(* PLC project CHL-DZ-BJDX-11 宁波数字孪生（东方理工）研究院制备薄层色谱全自动化工作站_Old_InoProShop(V1.9.1.6).project, Inovance company InoProShop(V1.9.1.6) InoProShop(V1.9.1.6) *)
(* stored: creationDateTime 2026-06-16T17:56:22.3681085, modificationDateTime 2026-06-04T10:59:46 *)

PROGRAM PLC_Cyinder_气缸动作
  VAR
    cylinder_0 : FB_cylinder;
    cylinder_1 : FB_cylinder;
    cylinder_2 : FB_cylinder;
    cylinder_3 : FB_cylinder;
    cylinder_4 : FB_cylinder;
    cylinder_5 : FB_cylinder;
    cylinder_6 : FB_cylinder;
    cylinder_7 : FB_cylinder;
    cylinder_8 : FB_cylinder;
    cylinder_9 : FB_cylinder;
    cylinder_10 : FB_cylinder;
    cylinder_11 : FB_cylinder;
    cylinder_12 : FB_cylinder;
    cylinder_13 : FB_cylinder;
    cylinder_14 : FB_cylinder;
    cylinder_15 : FB_cylinder;
    cylinder_16 : FB_cylinder;
    cylinder_17 : FB_cylinder;
    cylinder_18 : FB_cylinder;
    cylinder_19 : FB_cylinder;
    cylinder_20 : FB_cylinder;
    cylinder_21 : FB_cylinder;
    cylinder_22 : FB_cylinder;
    cylinder_23 : FB_cylinder;
    cylinder_24 : FB_cylinder;
    cylinder_25 : FB_cylinder;
    cylinder_26 : FB_cylinder;
    cylinder_27 : FB_cylinder;
    cylinder_28 : FB_cylinder;
    cylinder_29 : FB_cylinder;
    cylinder_30 : FB_cylinder;
    cylinder_31 : FB_cylinder;
    cylinder_32 : FB_cylinder;
    cylinder_33 : FB_cylinder;
    cylinder_34 : FB_cylinder;
    cylinder_35 : FB_cylinder;
    cylinder_36 : FB_cylinder;
    cylinder_37 : FB_cylinder;
    cylinder_38 : FB_cylinder;
    cylinder_39 : FB_cylinder;
    cylinder_40 : FB_cylinder;
    cylinder_41 : FB_cylinder;
    cylinder_42 : FB_cylinder;
    cylinder_43 : FB_cylinder;
    cylinder_44 : FB_cylinder;
    cylinder_45 : FB_cylinder;
    cylinder_46 : FB_cylinder;
    cylinder_47 : FB_cylinder;
    cylinder_48 : FB_cylinder;
    cylinder_49 : FB_cylinder;
    cylinder_50 : FB_cylinder;
  END_VAR

            //气缸动作
//展缸1气缸1
cylinder_0(
    xManualRetract := , 
    xAutoRetract := , 
    yValve2 => , 
    cylinder_type := 0, 

	xManualAuto:=ManualAuto  , 
	xManualExtend:=展缸1气缸1手动 , 
	xAutoExtend:= 展缸1气缸1自动, 
	xReset:=复位  , 
	xPosExtend:= 展缸1气缸1原点, 
	xPosRetract:= 展缸1气缸1动点 , 
	tTimeout:= T#5S, 
	yValve1=> 展缸1气缸1 , 
	bAlarm=> cyinderAlarm.0);
//展缸1气缸2
cylinder_1(
    xManualRetract := , 
    xAutoRetract := , 
    yValve2 => , 
    cylinder_type :=0 , 

	xManualAuto:=ManualAuto  , 
	xManualExtend:=展缸1气缸2手动 , 
	xAutoExtend:= 展缸1气缸2自动, 
	xReset:=复位  , 
	xPosExtend:= 展缸1气缸2原点, 
	xPosRetract:= 展缸1气缸2动点 , 
	tTimeout:= T#5S, 
	yValve1=> 展缸1气缸2, 
	bAlarm=> cyinderAlarm.1);
//展缸1气缸3
cylinder_2(
    xManualRetract := , 
    xAutoRetract := , 
    yValve2 => , 
    cylinder_type := 0, 

	xManualAuto:=ManualAuto  , 
	xManualExtend:=展缸1气缸3手动 , 
	xAutoExtend:= 展缸1气缸3自动, 
	xReset:=复位  , 
	xPosExtend:= 展缸1气缸3原点, 
	xPosRetract:= 展缸1气缸3动点 , 
	tTimeout:= T#5S, 
	yValve1=> 展缸1气缸3, 
	bAlarm=> cyinderAlarm.2);
//展缸1气缸4
cylinder_3(
    xManualRetract := , 
    xAutoRetract := , 
    yValve2 => , 
    cylinder_type :=0 , 

	xManualAuto:=ManualAuto  , 
	xManualExtend:=展缸1气缸4手动 , 
	xAutoExtend:= 展缸1气缸4自动, 
	xReset:=复位  , 
	xPosExtend:= 展缸1气缸4原点, 
	xPosRetract:= 展缸1气缸4动点 , 
	tTimeout:= T#5S, 
	yValve1=> 展缸1气缸4, 
	bAlarm=> cyinderAlarm.3);
//展缸2气缸1
cylinder_4(
    xManualRetract := , 
    xAutoRetract := , 
    yValve2 => , 
    cylinder_type := 0, 

	xManualAuto:=ManualAuto  , 
	xManualExtend:=展缸2气缸1手动 , 
	xAutoExtend:= 展缸2气缸1自动, 
	xReset:=复位  , 
	xPosExtend:= 展缸2气缸1原点, 
	xPosRetract:= 展缸2气缸1动点 , 
	tTimeout:= T#5S, 
	yValve1=> 展缸2气缸1, 
	bAlarm=> cyinderAlarm.4);
//展缸2气缸2
cylinder_5(
    xManualRetract := , 
    xAutoRetract := , 
    yValve2 => , 
    cylinder_type :=0 , 

	xManualAuto:=ManualAuto  , 
	xManualExtend:=展缸2气缸2手动 , 
	xAutoExtend:= 展缸2气缸2自动, 
	xReset:=复位  , 
	xPosExtend:= 展缸2气缸2原点, 
	xPosRetract:= 展缸2气缸2动点 , 
	tTimeout:= T#5S, 
	yValve1=> 展缸2气缸2, 
	bAlarm=> cyinderAlarm.5);
//展缸2气缸3
cylinder_6(
    xManualRetract := , 
    xAutoRetract := , 
    yValve2 => , 
    cylinder_type := 0, 

	xManualAuto:=ManualAuto  , 
	xManualExtend:=展缸2气缸3手动 , 
	xAutoExtend:= 展缸2气缸3自动, 
	xReset:=复位  , 
	xPosExtend:= 展缸2气缸3原点, 
	xPosRetract:= 展缸2气缸3动点 , 
	tTimeout:= T#5S, 
	yValve1=> 展缸2气缸3, 
	bAlarm=> cyinderAlarm.6);
//展缸2气缸4
cylinder_7(
    xManualRetract := , 
    xAutoRetract := , 
    yValve2 => , 
    cylinder_type := 0, 

	xManualAuto:=ManualAuto  , 
	xManualExtend:=展缸2气缸4手动 , 
	xAutoExtend:= 展缸2气缸4自动, 
	xReset:=复位  , 
	xPosExtend:= 展缸2气缸4原点, 
	xPosRetract:= 展缸2气缸4动点 , 
	tTimeout:= T#5S, 
	yValve1=> 展缸2气缸4, 
	bAlarm=> cyinderAlarm.7);
//大真空泵
cylinder_8(
    xManualRetract := , 
    xAutoRetract := , 
    yValve2 => , 
    cylinder_type :=0 , 

	xManualAuto:=ManualAuto  , 
	xManualExtend:= 大真空泵手动, 
	xAutoExtend:= 大真空泵自动, 
	xReset:=复位  , 
	xPosExtend:= , 
	xPosRetract:=  , 
	tTimeout:= , 
	yValve1=> 大真空泵, 
	bAlarm=> );
//收集平台下压气缸
cylinder_9(
    xManualRetract := , 
    xAutoRetract := , 
    yValve2 => , 
    cylinder_type := 0, 

	xManualAuto:=ManualAuto  , 
	xManualExtend:= 收集下压气缸手动, 
	xAutoExtend:= 收集下压气缸自动, 
	xReset:=复位  , 
	xPosExtend:=收集平台下压气缸原点 , 
	xPosRetract:= 收集下压气缸手动 OR 收集下压气缸自动, 
	tTimeout:= T#5S, 
	yValve1=> 收集下压气缸 , 
	bAlarm=> cyinderAlarm.8);
//收集平台夹持气缸
cylinder_10(
    xManualRetract := , 
    xAutoRetract := , 
    yValve2 => , 
    cylinder_type := 0, 

	xManualAuto:=ManualAuto  , 
	xManualExtend:= 收集夹持气缸手动, 
	xAutoExtend:= 收集夹持气缸自动, 
	xReset:=复位  , 
	xPosExtend:=收集平台夹持气缸原点 , 
	xPosRetract:= 收集平台夹持气缸动点, 
	tTimeout:= T#5S, 
	yValve1=> 收集夹持气缸  , 
	bAlarm=> cyinderAlarm.9);	
//收集平台升降气缸
cylinder_11(
    xManualRetract := , 
    xAutoRetract := , 
    yValve2 => , 
    cylinder_type := 0, 

	xManualAuto:=ManualAuto  , 
	xManualExtend:= 收集升降气缸手动, 
	xAutoExtend:= 收集升降气缸自动, 
	xReset:=复位  , 
	xPosExtend:=收集平台升降气缸原点 , 
	xPosRetract:= 收集平台升降气缸动点, 
	tTimeout:= T#5S, 
	yValve1=> 收集升降气缸   , 
	bAlarm=> cyinderAlarm.10);	
//收集平台伸缩气缸
cylinder_12(
    xManualRetract := , 
    xAutoRetract := , 
    yValve2 => , 
    cylinder_type :=0 , 

	xManualAuto:=ManualAuto  , 
	xManualExtend:= 收集伸缩气缸手动, 
	xAutoExtend:= 收集伸缩气缸自动, 
	xReset:=复位, 
	xPosExtend:=收集平台推出气缸原点, 
	xPosRetract:= 收集平台推出气缸动点, 
	tTimeout:= T#5S, 
	yValve1=> 收集伸缩气缸, 
	bAlarm=> cyinderAlarm.11);		
//刮板拍照遮光气缸
cylinder_13(
    xManualRetract := , 
    xAutoRetract := , 
    yValve2 => , 
    cylinder_type :=0 , 

	xManualAuto:=ManualAuto  , 
	xManualExtend:= 刮板拍照遮光气缸手动, 
	xAutoExtend:=刮板拍照遮光气缸自动 , 
	xReset:=复位  , 
	xPosExtend:=刮板拍照遮光气缸上位 , 
	xPosRetract:= 刮板拍照遮光气缸下位, 
	tTimeout:= T#5S, 
	yValve1=>  刮板拍照遮光气缸, 
	bAlarm=> cyinderAlarm.12);		
//刮板拍照旋转气缸
cylinder_14(
    xManualRetract := , 
    xAutoRetract := , 
    yValve2 => , 
    cylinder_type := 0, 

	xManualAuto:=ManualAuto  , 
	xManualExtend:= 刮板拍照旋转气缸手动 AND 刮板轴9XDATE.fActPos>330, 
	xAutoExtend:=刮板拍照旋转气缸自动 , 
	xReset:=复位  , 
	xPosExtend:=刮板拍照旋转气缸原点  , 
	xPosRetract:= 刮板拍照旋转气缸动点, 
	tTimeout:= T#5S, 
	yValve1=>  刮板拍照旋转气缸   , 
	bAlarm=> cyinderAlarm.13);		
//刮板拍照下压气缸
cylinder_15(
    xManualRetract := , 
    xAutoRetract := , 
    yValve2 => , 
    cylinder_type := 0, 

	xManualAuto:=ManualAuto  , 
	xManualExtend:= 刮板拍照下压气缸手动, 
	xAutoExtend:=刮板拍照下压气缸自动 , 
	xReset:=复位  , 
	xPosExtend:=刮板拍照下压气缸上位, 
	xPosRetract:=刮板拍照下压气缸手动 OR 刮板拍照下压气缸自动 , 
	tTimeout:= T#5S, 
	yValve1=>  刮板拍照下压气缸, 
	bAlarm=> cyinderAlarm.14);
//展缸1进液电池阀1
cylinder_17(
    xManualRetract := , 
    xAutoRetract := , 
    yValve2 => , 
    cylinder_type :=0 , 

	xManualAuto:=ManualAuto  , 
	xManualExtend:= 展缸1进液电池阀1手动, 
	xAutoExtend:= 展缸1进液电池阀1自动, 
	xReset:=复位  , 
	xPosExtend:=   , 
	xPosRetract:= , 
	tTimeout:= , 
	yValve1=> 展缸1进液电池阀1, 
	bAlarm=> );	
//展缸1进液电池阀2
cylinder_18(
    xManualRetract := , 
    xAutoRetract := , 
    yValve2 => , 
    cylinder_type := 0, 

	xManualAuto:=ManualAuto  , 
	xManualExtend:= 展缸1进液电池阀2手动, 
	xAutoExtend:= 展缸1进液电池阀2自动, 
	xReset:=复位  , 
	xPosExtend:=   , 
	xPosRetract:= , 
	tTimeout:= , 
	yValve1=> 展缸1进液电池阀2, 
	bAlarm=> );	
//展缸1进液电池阀3
cylinder_19(
    xManualRetract := , 
    xAutoRetract := , 
    yValve2 => , 
    cylinder_type := 0, 

	xManualAuto:=ManualAuto  , 
	xManualExtend:= 展缸1进液电池阀3手动, 
	xAutoExtend:= 展缸1进液电池阀3自动, 
	xReset:=复位  , 
	xPosExtend:=   , 
	xPosRetract:= , 
	tTimeout:= , 
	yValve1=> 展缸1进液电池阀3, 
	bAlarm=> );	
//展缸1进液电池阀4
cylinder_20(
    xManualRetract := , 
    xAutoRetract := , 
    yValve2 => , 
    cylinder_type := 0, 

	xManualAuto:=ManualAuto  , 
	xManualExtend:= 展缸1进液电池阀4手动, 
	xAutoExtend:= 展缸1进液电池阀4自动, 
	xReset:=复位  , 
	xPosExtend:=   , 
	xPosRetract:= , 
	tTimeout:= , 
	yValve1=> 展缸1进液电池阀4, 
	bAlarm=> );	
//展缸1排液电池阀1
cylinder_21(
    xManualRetract := , 
    xAutoRetract := , 
    yValve2 => , 
    cylinder_type := 0, 

	xManualAuto:=ManualAuto  , 
	xManualExtend:= 展缸1排液电池阀1手动, 
	xAutoExtend:= 展缸1排液电池阀1自动, 
	xReset:=复位  , 
	xPosExtend:=   , 
	xPosRetract:= , 
	tTimeout:= , 
	yValve1=> 展缸1排液电池阀1, 
	bAlarm=> );	
//展缸1排液电池阀2
cylinder_22(
    xManualRetract := , 
    xAutoRetract := , 
    yValve2 => , 
    cylinder_type :=0 , 

	xManualAuto:=ManualAuto  , 
	xManualExtend:= 展缸1排液电池阀2手动, 
	xAutoExtend:= 展缸1排液电池阀2自动, 
	xReset:=复位  , 
	xPosExtend:=   , 
	xPosRetract:= , 
	tTimeout:= , 
	yValve1=> 展缸1排液电池阀2, 
	bAlarm=> );	
//展缸1排液电池阀3
cylinder_23(
    xManualRetract := , 
    xAutoRetract := , 
    yValve2 => , 
    cylinder_type :=0 , 

	xManualAuto:=ManualAuto, 
	xManualExtend:= 展缸1排液电池阀3手动, 
	xAutoExtend:= 展缸1排液电池阀3自动, 
	xReset:=复位  , 
	xPosExtend:=   , 
	xPosRetract:= , 
	tTimeout:= , 
	yValve1=> 展缸1排液电池阀3, 
	bAlarm=> );	
//展缸1排液电池阀4
cylinder_24(
    xManualRetract := , 
    xAutoRetract := , 
    yValve2 => , 
    cylinder_type := 0, 

	xManualAuto:=ManualAuto, 
	xManualExtend:= 展缸1排液电池阀4手动, 
	xAutoExtend:= 展缸1排液电池阀4自动, 
	xReset:=复位  , 
	xPosExtend:=   , 
	xPosRetract:= , 
	tTimeout:= , 
	yValve1=> 展缸1排液电池阀4, 
	bAlarm=> );	
//展缸1吹气电池阀1
cylinder_25(
    xManualRetract := , 
    xAutoRetract := , 
    yValve2 => , 
    cylinder_type := 0, 

	xManualAuto:=ManualAuto, 
	xManualExtend:= 展缸1吹气电池阀1手动, 
	xAutoExtend:= 展缸1吹气电池阀1自动, 
	xReset:=复位  , 
	xPosExtend:=   , 
	xPosRetract:= , 
	tTimeout:= , 
	yValve1=> 展缸1吹气电池阀1, 
	bAlarm=> );	
//展缸1吹气电池阀2
cylinder_26(
    xManualRetract := , 
    xAutoRetract := , 
    yValve2 => , 
    cylinder_type := 0, 

	xManualAuto:=ManualAuto, 
	xManualExtend:= 展缸1吹气电池阀2手动, 
	xAutoExtend:= 展缸1吹气电池阀2自动, 
	xReset:=复位  , 
	xPosExtend:=   , 
	xPosRetract:= , 
	tTimeout:= , 
	yValve1=> 展缸1吹气电池阀2, 
	bAlarm=> );	
//展缸1吹气电池阀3
cylinder_27(
    xManualRetract := , 
    xAutoRetract := , 
    yValve2 => , 
    cylinder_type := 0, 

	xManualAuto:=ManualAuto  , 
	xManualExtend:= 展缸1吹气电池阀3手动, 
	xAutoExtend:= 展缸1吹气电池阀3自动, 
	xReset:=复位  , 
	xPosExtend:=   , 
	xPosRetract:= , 
	tTimeout:= , 
	yValve1=> 展缸1吹气电池阀3, 
	bAlarm=> );	
//展缸1吹气电池阀4
cylinder_28(
    xManualRetract := , 
    xAutoRetract := , 
    yValve2 => , 
    cylinder_type := 0, 

	xManualAuto:=ManualAuto, 
	xManualExtend:= 展缸1吹气电池阀4手动, 
	xAutoExtend:= 展缸1吹气电池阀4自动, 
	xReset:=复位  , 
	xPosExtend:=   , 
	xPosRetract:= , 
	tTimeout:= , 
	yValve1=> 展缸1吹气电池阀4, 
	bAlarm=> );	
//展缸2进液电池阀1
cylinder_29(
    xManualRetract := , 
    xAutoRetract := , 
    yValve2 => , 
    cylinder_type := 0, 

	xManualAuto:=ManualAuto, 
	xManualExtend:= 展缸2进液电池阀1手动, 
	xAutoExtend:= 展缸2进液电池阀1自动, 
	xReset:=复位  , 
	xPosExtend:=   , 
	xPosRetract:= , 
	tTimeout:= , 
	yValve1=> 展缸2进液电池阀1, 
	bAlarm=> );	
//展缸2进液电池阀2
cylinder_30(
    xManualRetract := , 
    xAutoRetract := , 
    yValve2 => , 
    cylinder_type := 0, 

	xManualAuto:=ManualAuto, 
	xManualExtend:= 展缸2进液电池阀2手动, 
	xAutoExtend:= 展缸2进液电池阀2自动, 
	xReset:=复位  , 
	xPosExtend:=   , 
	xPosRetract:= , 
	tTimeout:= , 
	yValve1=> 展缸2进液电池阀2, 
	bAlarm=> );	
//展缸2进液电池阀3
cylinder_31(
    xManualRetract := , 
    xAutoRetract := , 
    yValve2 => , 
    cylinder_type := 0, 

	xManualAuto:=ManualAuto, 
	xManualExtend:= 展缸2进液电池阀3手动, 
	xAutoExtend:= 展缸2进液电池阀3自动, 
	xReset:=复位  , 
	xPosExtend:=   , 
	xPosRetract:= , 
	tTimeout:= , 
	yValve1=> 展缸2进液电池阀3, 
	bAlarm=> );	
//展缸2进液电池阀4
cylinder_32(
    xManualRetract := , 
    xAutoRetract := , 
    yValve2 => , 
    cylinder_type := 0, 

	xManualAuto:=ManualAuto, 
	xManualExtend:= 展缸2进液电池阀4手动, 
	xAutoExtend:= 展缸2进液电池阀4自动, 
	xReset:=复位  , 
	xPosExtend:=   , 
	xPosRetract:= , 
	tTimeout:= , 
	yValve1=> 展缸2进液电池阀4, 
	bAlarm=> );	
//展缸2排液电池阀1
cylinder_33(
    xManualRetract := , 
    xAutoRetract := , 
    yValve2 => , 
    cylinder_type := 0, 

	xManualAuto:=ManualAuto, 
	xManualExtend:= 展缸2排液电池阀1手动, 
	xAutoExtend:= 展缸2排液电池阀1自动, 
	xReset:=复位  , 
	xPosExtend:=   , 
	xPosRetract:= , 
	tTimeout:= , 
	yValve1=> 展缸2排液电池阀1, 
	bAlarm=> );	
//展缸2排液电池阀2
cylinder_34(
    xManualRetract := , 
    xAutoRetract := , 
    yValve2 => , 
    cylinder_type := 0, 

	xManualAuto:=ManualAuto, 
	xManualExtend:= 展缸2排液电池阀2手动, 
	xAutoExtend:= 展缸2排液电池阀2自动, 
	xReset:=复位  , 
	xPosExtend:=   , 
	xPosRetract:= , 
	tTimeout:= , 
	yValve1=> 展缸2排液电池阀2, 
	bAlarm=> );	
//展缸2排液电池阀3
cylinder_35(
    xManualRetract := , 
    xAutoRetract := , 
    yValve2 => , 
    cylinder_type := 0, 

	xManualAuto:=ManualAuto, 
	xManualExtend:= 展缸2排液电池阀3手动, 
	xAutoExtend:= 展缸2排液电池阀3自动, 
	xReset:=复位  , 
	xPosExtend:=   , 
	xPosRetract:= , 
	tTimeout:= , 
	yValve1=> 展缸2排液电池阀3, 
	bAlarm=> );	
//展缸2排液电池阀4
cylinder_36(
    xManualRetract := , 
    xAutoRetract := , 
    yValve2 => , 
    cylinder_type :=0 , 

	xManualAuto:=ManualAuto, 
	xManualExtend:= 展缸2排液电池阀4手动, 
	xAutoExtend:= 展缸2排液电池阀4自动, 
	xReset:=复位  , 
	xPosExtend:=   , 
	xPosRetract:= , 
	tTimeout:= , 
	yValve1=> 展缸2排液电池阀4, 
	bAlarm=> );	
//展缸2吹气电池阀1
cylinder_37(
    xManualRetract := , 
    xAutoRetract := , 
    yValve2 => , 
    cylinder_type := 0, 

	xManualAuto:=ManualAuto, 
	xManualExtend:= 展缸2吹气电池阀1手动, 
	xAutoExtend:= 展缸2吹气电池阀1自动, 
	xReset:=复位  , 
	xPosExtend:=   , 
	xPosRetract:= , 
	tTimeout:= , 
	yValve1=> 展缸2吹气电池阀1, 
	bAlarm=> );	
//展缸2吹气电池阀2
cylinder_38(
    xManualRetract := , 
    xAutoRetract := , 
    yValve2 => , 
    cylinder_type := 0, 

	xManualAuto:=ManualAuto, 
	xManualExtend:= 展缸2吹气电池阀2手动, 
	xAutoExtend:= 展缸2吹气电池阀2自动, 
	xReset:=复位  , 
	xPosExtend:=   , 
	xPosRetract:= , 
	tTimeout:= , 
	yValve1=> 展缸2吹气电池阀2, 
	bAlarm=> );	
//展缸1吹气电池阀3
cylinder_39(
    xManualRetract := , 
    xAutoRetract := , 
    yValve2 => , 
    cylinder_type := 0, 

	xManualAuto:=ManualAuto, 
	xManualExtend:= 展缸2吹气电池阀3手动, 
	xAutoExtend:= 展缸2吹气电池阀3自动, 
	xReset:=复位  , 
	xPosExtend:=   , 
	xPosRetract:= , 
	tTimeout:= , 
	yValve1=> 展缸2吹气电池阀3, 
	bAlarm=> );	
//展缸2吹气电池阀4
cylinder_40(
    xManualRetract := , 
    xAutoRetract := , 
    yValve2 => , 
    cylinder_type := 0, 

	xManualAuto:=ManualAuto, 
	xManualExtend:= 展缸2吹气电池阀4手动, 
	xAutoExtend:= 展缸2吹气电池阀4自动, 
	xReset:=复位  , 
	xPosExtend:=   , 
	xPosRetract:= , 
	tTimeout:= , 
	yValve1=> 展缸2吹气电池阀4, 
	bAlarm=> );	
//收集进液电池阀
cylinder_41(
    xManualRetract := , 
    xAutoRetract := , 
    yValve2 => , 
    cylinder_type := 0, 

	xManualAuto:=ManualAuto, 
	xManualExtend:= 收集进液手动, 
	xAutoExtend:= 收集进液自动, 
	xReset:=复位  , 
	xPosExtend:=   , 
	xPosRetract:= , 
	tTimeout:= , 
	yValve1=> 收集平台进液2通电池阀, 
	bAlarm=> );	
//收集排液电池阀
cylinder_42(
    xManualRetract := , 
    xAutoRetract := , 
    yValve2 => , 
    cylinder_type := 0, 

	xManualAuto:=ManualAuto  , 
	xManualExtend:= 收集排液手动, 
	xAutoExtend:= 收集排液自动, 
	xReset:=复位  , 
	xPosExtend:=   , 
	xPosRetract:= , 
	tTimeout:= , 
	yValve1=> 收集平台排液3通电池阀, 
	bAlarm=> );	
//收集正压排液电池阀
cylinder_43(
    xManualRetract := , 
    xAutoRetract := , 
    yValve2 => , 
    cylinder_type :=0 , 

	xManualAuto:=ManualAuto  , 
	xManualExtend:= 收集正压排液手动, 
	xAutoExtend:= 收集正压排液自动, 
	xReset:=复位  , 
	xPosExtend:=   , 
	xPosRetract:= , 
	tTimeout:= , 
	yValve1=> 收集平台正压排液阀, 
	bAlarm=> );	
//溶液收集瓶定位气缸
cylinder_44(
    xManualRetract := , 
    xAutoRetract := , 
    yValve2 => , 
    cylinder_type := 0, 

	xManualAuto:=ManualAuto  , 
	xManualExtend:= 溶液收集瓶定位手动, 
	xAutoExtend:= 溶液收集瓶定位自动, 
	xReset:=复位  , 
	xPosExtend:=   , 
	xPosRetract:= , 
	tTimeout:= , 
	yValve1=> 溶液收集瓶工位定位气缸, 
	bAlarm=> );	
//上样定位气缸
cylinder_45(
    xManualRetract := , 
    xAutoRetract := , 
    yValve2 => , 
    cylinder_type :=0 , 

	xManualAuto:=ManualAuto  , 
	xManualExtend:= 上样定位手动, 
	xAutoExtend:= 上样定位自动, 
	xReset:=复位  , 
	xPosExtend:=   , 
	xPosRetract:= , 
	tTimeout:= , 
	yValve1=> 上样定位气缸, 
	bAlarm=> );	
//上样点样三通电池阀
cylinder_46(
    xManualRetract := , 
    xAutoRetract := , 
    yValve2 => , 
    cylinder_type :=0 , 

	xManualAuto:=ManualAuto  , 
	xManualExtend:= 上样点样三通电池阀手动, 
	xAutoExtend:= 上样点样三通电池阀自动, 
	xReset:=复位  , 
	xPosExtend:=   , 
	xPosRetract:= , 
	tTimeout:= , 
	yValve1=> 上样点样三通电池阀, 
	bAlarm=> );	
//刮板拍照真空泵
cylinder_46(
    xManualRetract := , 
    xAutoRetract := , 
    yValve2 => , 
    cylinder_type := 0, 

	xManualAuto:=ManualAuto  , 
	xManualExtend:=刮板拍照真空手动 , 
	xAutoExtend:= 刮板拍照真空自动, 
	xReset:=复位  , 
	xPosExtend:=   , 
	xPosRetract:= , 
	tTimeout:= , 
	yValve1=> 刮板拍照真空阀, 
	bAlarm=> );	
//刮板拍照无刷电机
cylinder_47(
    xManualRetract := , 
    xAutoRetract := , 
    yValve2 => , 
    cylinder_type :=0 , 

	xManualAuto:=ManualAuto  , 
	xManualExtend:=刮板拍照无刷电机手动 , 
	xAutoExtend:=刮板拍照无刷电机自动 , 
	xReset:=复位  , 
	xPosExtend:=   , 
	xPosRetract:= , 
	tTimeout:= , 
	yValve1=> 刮板拍照无刷电机, 
	bAlarm=> );	
//刮板拍照定位气缸
cylinder_48(
    xManualRetract := , 
    xAutoRetract := , 
    yValve2 => , 
    cylinder_type :=0 , 

	xManualAuto:=ManualAuto  , 
	xManualExtend:= 刮板拍照定位气缸手动, 
	xAutoExtend:=刮板拍照定位气缸自动 , 
	xReset:=复位  , 
	xPosExtend:=   , 
	xPosRetract:= , 
	tTimeout:= , 
	yValve1=> 刮板拍照定位气缸, 
	bAlarm=> );	
//粉末收集器定位气缸
cylinder_49(
    xManualRetract := , 
    xAutoRetract := , 
    yValve2 => , 
    cylinder_type :=0 , 

	xManualAuto:=ManualAuto  , 
	xManualExtend:= 粉末收集器定位手动, 
	xAutoExtend:= 粉末收集器定位自动, 
	xReset:=复位  , 
	xPosExtend:=   , 
	xPosRetract:= , 
	tTimeout:= , 
	yValve1=> 粉末收集器工位定位气缸, 
	bAlarm=> );	
//上样吹气电池阀
cylinder_50(
    xManualRetract := , 
    xAutoRetract := , 
    yValve2 => , 
    cylinder_type := 0, 

	xManualAuto:=ManualAuto  , 
	xManualExtend:= 上样吹气手动, 
	xAutoExtend:= 上样吹气自动, 
	xReset:=复位  , 
	xPosExtend:=   , 
	xPosRetract:= , 
	tTimeout:= , 
	yValve1=> 上样吹气二通阀, 
	bAlarm=> );	








	
	
          
END_PROGRAM
